# EPICS substitutions: pacman-softIoc/game_engine.subs
file pacman_game_parameter.template
{ pattern
  { NAME,	DEVICE,	P,	DRVH,	DRVL,	VAL	}
  { GAME, STATE, INDICATOR, 10, 0, 0 }
  { GAME, KILLED, GHOSTS_MULTIPLIER, 100, 0, 1 }
  { GAME, WIN, CONDITION, 244, 0, 244 }
}

file pacman_binary_records.template
{ pattern
  { NAME,	DEVICE,	P, ZNAM, ONAM,	VAL,	HIGH }
  { GAME, FRIGHT, MODE, DISABLED, ENABLED, 0, 20 }
  { GAME, GHOSTS, INKY_RELEASE, RELEASED, WAITING, 0, 7 }
  { GAME, GHOSTS, CLYDE_RELEASE, RELEASED, WAITING, 0, 7 }
  { GAME, GHOSTS, BLINKY_RESPAWN, DONE, WAITING, 0, 5 }
  { GAME, GHOSTS, PINKY_RESPAWN, DONE, WAITING, 0, 5 }
  { GAME, GHOSTS, INKY_RESPAWN, DONE, WAITING, 0, 5 }
  { GAME, GHOSTS, CLYDE_RESPAWN, DONE, WAITING, 0, 5 }
}
